PROGRAM CreateJsonDocumentAuto
VAR_INPUT
	visionFrameData : REFERENCE TO VisionFrame;
END_VAR
VAR_OUTPUT
	jsonDocument : STRING(1000); 
END_VAR
VAR
	fbJson : FB_JsonSaxWriter;
	fbJsonDataType : FB_JsonReadWriteDataType;
END_VAR

fbJson.ResetDocument();

fbJsonDataType.AddJsonValueFromSymbol(fbJson, 'VisionFrame', SIZEOF(visionFrameData), ADR(visionFrameData));

fbJson.CopyDocument(jsonDocument, SIZEOF(jsonDocument));

END_PROGRAM

(* stored: Version 1.1.0.1, ProductVersion 3.1.4024.11
   POU CreateJsonDocumentAuto: Id {4213c277-03d4-4979-8ce4-3c9baf2d9087}, SpecialFunc None *)
